RoboDK station: Final ChArUco Hand-Eye Calibration.rdk

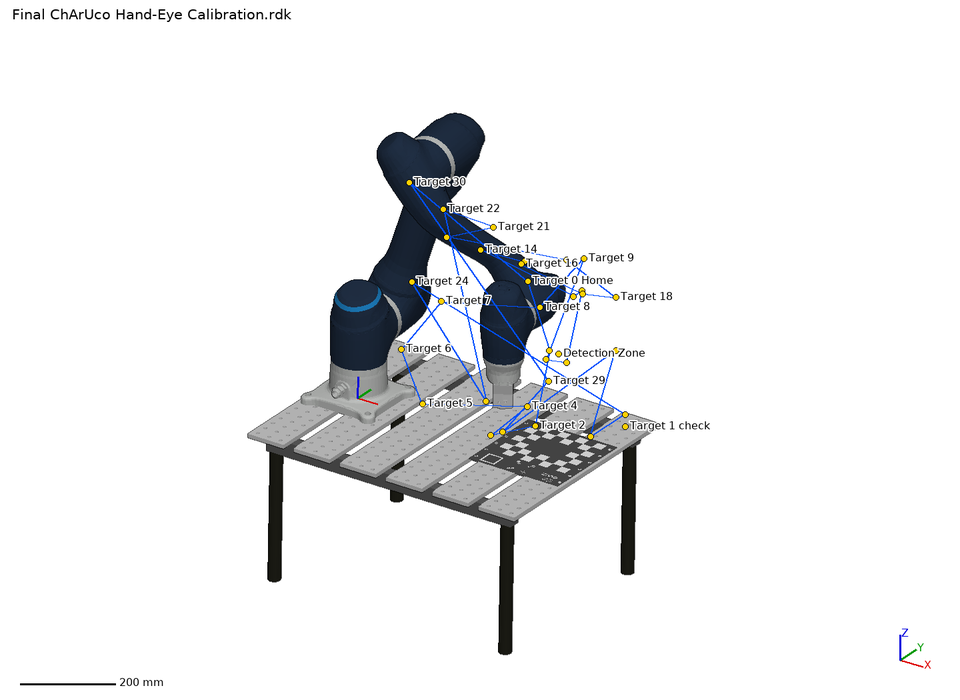
[picture v0: the station drawn from its stored meshes, robots at their saved joint values, targets as dots, program paths as lines]
Station Final ChArUco Hand-Eye Calibration (saved by RoboDK 5.9.2). Poses are relative to the parent item; angles as X-Y-Z fixed-axis rotations.
Station parameters (name, value as stored): IO_2, 0, IO_5, 1, IO_3, 0, 2, 0, 3, 0
  - program declamping (2 instructions, listed below)
  - program clamping (2 instructions, listed below)
  - frame World at (141.88, -8.76, 0) mm, rotated rx 0 ry 1.07 rz 1.07 deg
    - frame Doosan Robotics A0509 Base at (0, 0, 0) mm
      - robot Doosan Robotics A0509: 6 axes, payload 5 kg, reach 900 mm, repeatability 0.03 mm
          modified DH rows (alpha deg, a mm, theta deg, d mm): 0, 0, 0, 155.5; -90, 0, -90, 0; 0, 409, -90, 0; -90, 0, 0, 367; 90, 0, 0, 0; -90, 0, 90, 124
          base shift (0, 0, 0) mm, rotated rx 0 ry 0 rz 180 deg
          joint limits [-360, -360, -150, -360, -360, -360] to [360, 360, 150, 360, 360, 360]; home [0, 0, 90, 0, 0, 0]; saved at [5.923, 16.954, 125.95, -0.003, 37.095, 63.023]
        - tool Camera Position, TCP at (0, 0, 45) mm, size 42 x 50.8 x 80 mm, geometry from World
      - target Target 1 check (Cartesian target) at (620.07, 75.01, 85.08) mm, rotated rx -180 ry -0.02 rz 0 deg; joints [6.34, 38.07, 89.434, -0.001, 52.478, -173.659] of Doosan Robotics A0509
    - target Detection Zone (Cartesian target) at (499.97, 0.1, 249.99) mm, rotated rx -180 ry 0 rz 0 deg; joints [-2.032, 11.28, 100.743, 0, 67.974, 177.968] of Doosan Robotics A0509
    - target Target 0 Home (Cartesian target) at (420, 0, 395.5) mm, rotated rx 180 ry 0 rz 0 deg; joints [0, 7.448, 82.013, 0, 90.539, 180] of Doosan Robotics A0509
    - target Target 1 (Cartesian target) at (476.93, 0, 249.96) mm, rotated rx 180 ry 0 rz 0 deg; joints [0.001, 8.187, 104.47, -0.003, 67.338, 180.001] of Doosan Robotics A0509
    - target Target 2 (Cartesian target) at (584.73, -211.96, 191.89) mm, rotated rx -137.58 ry 27.04 rz -24.17 deg; joints [-30.572, 40.445, 69.864, 39.843, 98.921, 180] of Doosan Robotics A0509
    - target Target 3 (Cartesian target) at (474.75, -212.29, 138.34) mm, rotated rx 178.38 ry 45.91 rz -89.52 deg; joints [-30.068, 34.843, 84.14, 37.157, 90.198, 228.903] of Doosan Robotics A0509
    - target Target 4 (Cartesian target) at (551.04, -191.94, 219.34) mm, rotated rx -150.91 ry 21.54 rz -30.04 deg; joints [-27.19, 30.476, 78.926, 30.105, 90.539, 183.38] of Doosan Robotics A0509
    - target Target 5 (Cartesian target) at (354.8, -291.67, 208.8) mm, rotated rx -150.39 ry 35.58 rz -61.71 deg; joints [-50.202, 18.344, 99.052, 35.824, 91.564, 192.668] of Doosan Robotics A0509
    - target Target 6 (Cartesian target) at (227.5, -181.7, 254.33) mm, rotated rx 140.96 ry -15.06 rz 122.26 deg; joints [-59.376, 10.835, 111.611, 39.718, 77.465, -12.245] of Doosan Robotics A0509
    - target Target 7 (Cartesian target) at (263.7, -88.93, 338.9) mm, rotated rx 157.82 ry -33.21 rz 68.19 deg; joints [-54.472, -12.634, 123.141, 41.605, 71.777, 49.66] of Doosan Robotics A0509
    - target Target 8 (Cartesian target) at (429.5, 33.17, 323.91) mm, rotated rx 179.88 ry -15.95 rz 1.98 deg; joints [5.46, -6.49, 111.891, -1.26, 58.69, 184.003] of Doosan Robotics A0509
    - target Target 9 (Cartesian target) at (600.86, -62.78, 527.2) mm, rotated rx 178.96 ry 0.02 rz -18.39 deg; joints [-3.769, 31.662, 26.69, -1.179, 121.922, 194.003] of Doosan Robotics A0509
    - target Target 10 (Cartesian target) at (504, -52.27, 258.93) mm, rotated rx -161.96 ry -2.39 rz 4.22 deg; joints [-14.735, 13.481, 98.454, 18.676, 72.76, 154.35] of Doosan Robotics A0509
    - target Target 11 (Cartesian target) at (513.58, 10.97, 229.27) mm, rotated rx -179.18 ry 0.65 rz 0.64 deg; joints [1.01, 14.41, 100.14, 0.9, 66.1, 180.003] of Doosan Robotics A0509
    - target Target 12 (Cartesian target) at (421.58, 203.14, 291.52) mm, rotated rx -177.09 ry 31.69 rz 92.46 deg; joints [27.564, 17.592, 83.119, -27.134, 96.077, 117.058] of Doosan Robotics A0509
    - target Target 13 (Cartesian target) at (482.28, 79.84, 345.96) mm, rotated rx -170.57 ry -12.63 rz -152.2 deg; joints [15.451, 33.395, 57.514, -12.059, 99.23, -14.272] of Doosan Robotics A0509
    - target Target 14 (Cartesian target) at (201.07, 149.89, 344.48) mm, rotated rx 154.26 ry 15.71 rz 91.8 deg; joints [40.953, -28.702, 118.946, -28.141, 79.248, 128.303] of Doosan Robotics A0509
    - target Target 15 (Cartesian target) at (272.84, 208.79, 314.14) mm, rotated rx 160.33 ry -6.2 rz 46.61 deg; joints [47.096, -16.289, 119.58, -20.803, 71.86, 187.259] of Doosan Robotics A0509
    - target Target 16 (Cartesian target) at (313.73, 133.78, 350.06) mm, rotated rx -162.42 ry 9.67 rz -172.93 deg; joints [36.361, -4.655, 94.326, -19.989, 90.771, 30.592] of Doosan Robotics A0509
    - target Target 17 (Cartesian target) at (386.52, 257.75, 252.02) mm, rotated rx -131.78 ry -12.84 rz -159.7 deg; joints [50.116, 30.688, 76.173, -36.803, 106.82, 24.06] of Doosan Robotics A0509
    - target Target 18 (Cartesian target) at (406.46, 354.8, 209.87) mm, rotated rx -152 ry 42.65 rz 137.18 deg; joints [45.81, 39.799, 65.351, -39.246, 105.639, 99.57] of Doosan Robotics A0509
    - target Target 19 (Cartesian target) at (411.03, 159.98, 377.64) mm, rotated rx -160.05 ry 2.22 rz -177.12 deg; joints [24.665, 23.534, 65.061, -19.421, 96.651, 20.799] of Doosan Robotics A0509
    - target Target 20 (Cartesian target) at (95.04, 181.88, 329.99) mm, rotated rx -153.95 ry 40.94 rz 178.29 deg; joints [97.305, -9.984, 111.444, -33.669, 112.378, 105.44] of Doosan Robotics A0509
    - target Target 21 (Cartesian target) at (195.15, 206.73, 371.97) mm, rotated rx -179.5 ry -50.53 rz -26.1 deg; joints [83.66, -7.131, 120.18, -46.844, 89.067, 300.003] of Doosan Robotics A0509
    - target Target 22 (Cartesian target) at (52.31, 232.85, 360.92) mm, rotated rx 169.22 ry 39.27 rz 127.84 deg; joints [102.182, -5.557, 99.853, -28.864, 114.906, 145.039] of Doosan Robotics A0509
    - target Target 23 (Cartesian target) at (468.99, -224.2, 221.17) mm, rotated rx 142.66 ry -36.08 rz 133.82 deg; joints [-38.89, 47.298, 66.868, 41.593, 95.189, 12.449] of Doosan Robotics A0509
    - target Target 24 (Cartesian target) at (129.65, -0.01, 309.79) mm, rotated rx -179.99 ry 49.13 rz -179.99 deg; joints [0.004, -48.939, 130.05, -0.005, 49.759, 0.001] of Doosan Robotics A0509
    - target Target 25 (Cartesian target) at (663.85, 8.24, 153.22) mm, rotated rx 179.19 ry 45.04 rz 0.31 deg; joints [0.866, 61.81, 31.232, -0.569, 132.002, 180.01] of Doosan Robotics A0509
    - target Target 26 (Cartesian target) at (663.84, -121.81, 153.34) mm, rotated rx 179.19 ry 45.03 rz -29.69 deg; joints [-11.845, 64.27, 26.308, 15.91, 132.112, 203.599] of Doosan Robotics A0509
    - target Target 27 (Cartesian target) at (588.56, 82.36, 249.82) mm, rotated rx -144.64 ry -29.96 rz 176.59 deg; joints [13.201, 71.456, 11.706, -34.588, 129.491, 352.316] of Doosan Robotics A0509
    - target Target 28 (Cartesian target) at (557.08, -292.04, 202.36) mm, rotated rx 134.41 ry 23.34 rz -137.32 deg; joints [-28.85, 72.93, 6.54, 43.04, 134.21, -60.002] of Doosan Robotics A0509
    - target Target 29 (Cartesian target) at (556.96, -122.02, 252.25) mm, rotated rx 153.66 ry 14.98 rz -100.93 deg; joints [-8.806, 43.211, 52.161, 15.362, 110.605, 270.696] of Doosan Robotics A0509
    - target Target 30 (Cartesian target) at (194.44, -113.14, 606.63) mm, rotated rx -176.79 ry -19.73 rz -7.95 deg; joints [-59.2, -25.601, 79.912, 19.091, 114.359, -222.146] of Doosan Robotics A0509
    - object Table 1200x1000mm (Welding) at (240, 0, 0) mm, size 671.5 x 542.9 x 342.9 mm, geometry from Table-1200x1000mm-Welding.sld
      - object Zivid ZVDA-CB01 Calibration Board at (103.57, -98.2, 0.2) mm, size 225 x 225 x 1.5 mm, geometry from Zivid-ZVDA-CB01-Calibration-Board.sld
  - program Prog3 (65 instructions, listed below)
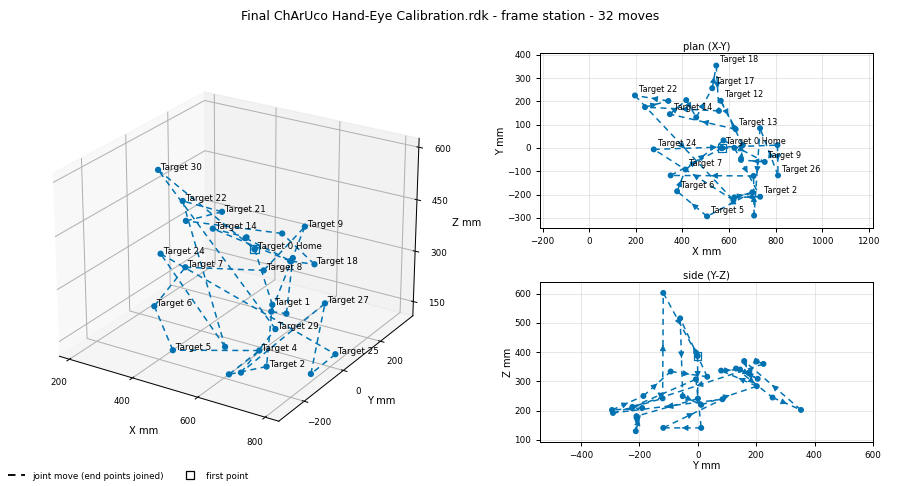
[picture p0: tool path of Final ChArUco Hand-Eye Calibration.rdk in frame station, 32 of 32 moves have a stored position in this frame; points joined in program order, loops and branches not executed]

--- program declamping (robot Doosan Robotics A0509) ---
  Set IO_2=1
  Set IO_2=0

--- program clamping (robot Doosan Robotics A0509) ---
  Set IO_3=1
  Set IO_3=0

--- program Prog3 (robot Doosan Robotics A0509) ---
  Set Ref.: World
  Set Tool: 560210_HGPT-35-A-B -> Camera Position
  MoveJ (Home Position) -> target Target 0 Home
  Pause 2.0 s
  MoveJ (Target 1)
  Pause 2.0 s
  MoveJ (Target 2)
  Pause 2.0 s
  MoveJ (Target 3)
  Pause 2.0 s
  MoveJ (Target 4)
  Pause 2.0 s
  MoveJ (Target 5)
  Pause 2.0 s
  MoveJ (Target 6)
  Pause 2.0 s
  MoveJ (Target 7)
  Pause 2.0 s
  MoveJ (Target 8)
  Pause 2.0 s
  MoveJ (Target 9)
  Pause 2.0 s
  MoveJ (Target 10)
  Pause 2.0 s
  MoveJ (Target 11)
  Pause 2.0 s
  MoveJ (Target 12)
  Pause 2.0 s
  MoveJ (Target 13)
  Pause 2.0 s
  MoveJ (Target 14)
  Pause 2.0 s
  MoveJ (Target 15)
  Pause 2.0 s
  MoveJ (Target 16)
  Pause 2.0 s
  MoveJ (Target 17)
  Pause 2.0 s
  MoveJ (Target 18)
  Pause 2.0 s
  MoveJ (Target 19)
  Pause 2.0 s
  MoveJ (Target 20)
  Pause 2.0 s
  MoveJ (Target 21)
  Pause 2.0 s
  MoveJ (Target 22)
  Pause 2.0 s
  MoveJ (Target 23)
  Pause 2.0 s
  MoveJ (Target 24)
  Pause 2.0 s
  MoveJ (Target 25)
  Pause 2.0 s
  MoveJ (Target 26)
  Pause 2.0 s
  MoveJ (Target 27)
  Pause 2.0 s
  MoveJ (Target 28)
  Pause 2.0 s
  MoveJ (Target 29)
  Pause 2.0 s
  MoveJ (Target 30)
  Pause 2.0 s
  MoveJ (Home Position) -> target Target 0 Home
